FUNCTION_BLOCK F_ABS (* absolute value *)
  PACKAGE iec61131::numerical;
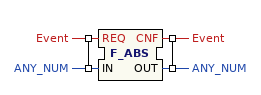
  EVENT_INPUT
    REQ WITH IN; (* Service Request *)
  END_EVENT
  EVENT_OUTPUT
    CNF WITH OUT; (* Confirmation of Requested Service *)
  END_EVENT
  VAR_INPUT
    IN : ANY_NUM; (* Event Input Qualifier *)
  END_VAR
  VAR_OUTPUT
    OUT : ANY_NUM; (* Event Output Qualifier *)
  END_VAR
END_FUNCTION_BLOCK
